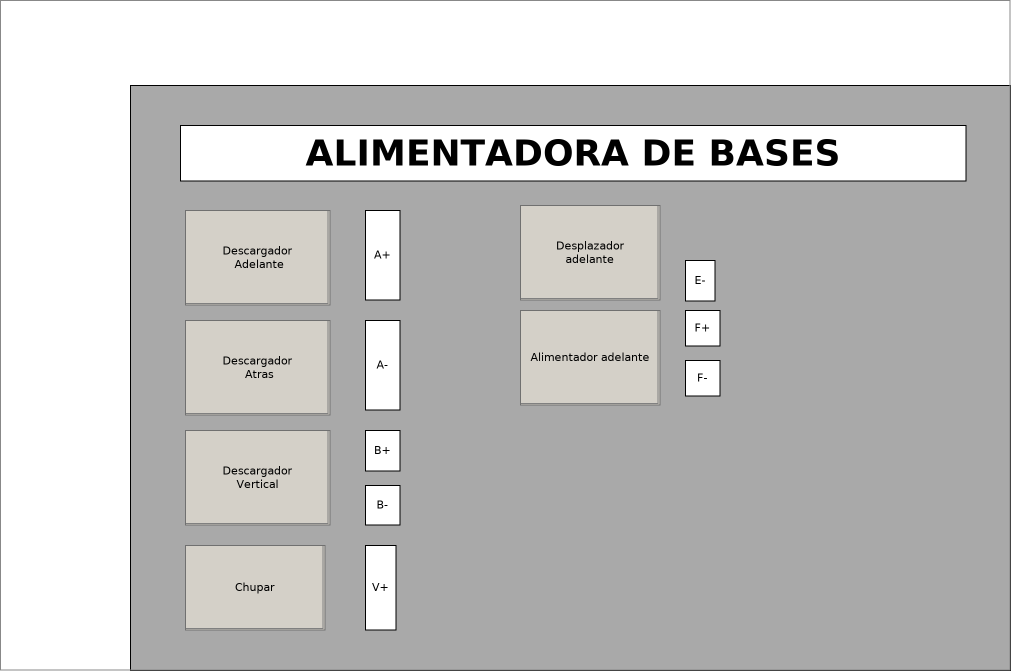
VISUALIZATION Visualization  // 1011x671
    Rectangle (130,85 881x586)
    Rectangle (180,125 786x56), "ALIMENTADORA DE BASES"
    Button (185,210 145x95), "Descargador Adelante", colour toggle: MAIN.ESTACION.DescargadorAdelante
        tap MAIN.ESTACION.DescargadorAdelante
    Button (185,320 145x95), "Descargador Atras", colour toggle: MAIN.ESTACION.DescargadorAtras
        tap MAIN.ESTACION.DescargadorAtras
    Rectangle (365,210 35x90), "A+", colour toggle: MAIN.ESTACION.DescargadorDelante
    Rectangle (365,320 35x90), "A-", colour toggle: MAIN.ESTACION.DescargadorDetras
    Button (185,430 145x95), "Descargador Vertical", colour toggle: MAIN.ESTACION.DescargadorBaja
        toggle MAIN.ESTACION.DescargadorBaja
    Rectangle (365,430 35x41), "B+", colour toggle: MAIN.ESTACION.VerticalArriba
    Rectangle (365,485 35x40), "B-", colour toggle: MAIN.ESTACION.VerticalAbajo
    Button (185,545 140x85), "Chupar"
        toggle MAIN.ESTACION.EyectorSucciona
    Rectangle (365,545 31x85), "V+", colour toggle: MAIN.ESTACION.EyectorSucciona
    Button (520,205 140x95), "Desplazador adelante"
        toggle MAIN.ESTACION.DesplazadorAdelante
    Rectangle (685,260 30x41), "E-", colour toggle: MAIN.ESTACION.DesplazadorDetras
    Button (520,310 140x95), "Alimentador adelante"
        tap MAIN.ESTACION.AlimentadorAdelante
    Rectangle (685,310 35x36), "F+", colour toggle: MAIN.ESTACION.AlimentadorDelante
    Rectangle (685,360 35x36), "F-", colour toggle: MAIN.ESTACION.AlimentadorDetras
END_VISUALIZATION

(* stored: Version 1.1.0.1, ProductVersion 3.1.4024.12
   Visu Visualization: Id {be50fb56-e4f5-4d7c-833b-55f83a8a37e1} *)
